FUNCTION WriteToInterlockAndLimit
VAR_INPUT
	value: BOOL;
	pos: DINT;
END_VAR
VAR
	BoolNumber : UDINT;
	result : UDINT;
END_VAR

BoolNumber := SHL(BOOL_TO_UDINT(value AND 1),pos);
result := DINT_TO_UDINT(Process.InterlockAndLimit) OR BoolNumber;
Process.InterlockAndLimit := UDINT_TO_DINT(result);

END_FUNCTION

(* stored: Version 1.1.0.1, ProductVersion 3.1.4024.9
   POU WriteToInterlockAndLimit: Id {b71cc806-851f-4f23-b41c-ed85b3044ef0}, SpecialFunc None *)
